// TwinCAT 3 PLC project OEF_6
// ProgramVersion: 3.1.4024.0
// libraries:
//   Tc2_BABasic, * (Beckhoff Automation GmbH)
//   Tc2_Standard, * (Beckhoff Automation GmbH)
//   Tc2_System, * (Beckhoff Automation GmbH)
//   Tc3_Module, * (Beckhoff Automation GmbH)
// project tree:
//   / PlcTask.TcTTO
//   POUs/ MAIN.TcPOU
// (motion and I/O tree: see PLC project oef_1)
// real-time tasks:
//   TASK PlcTask: cycle T#10ms, priority 20, ADS port 350
//   TASK PlcTask1: cycle T#10ms, priority 21, ADS port 351
//   TASK PlcTask2: cycle T#10ms, priority 22, ADS port 352
//   TASK PlcTask3: cycle T#10ms, priority 23, ADS port 353
//   TASK PlcTask4: cycle T#10ms, priority 24, ADS port 354
//   TASK PlcTask5: cycle T#10ms, priority 25, ADS port 355
//   TASK PlcTask6: cycle T#10ms, priority 26, ADS port 356
// variable links:
//   OEF_6/OEF_6 Instance <-> Device 1 (EtherCAT)/Term 1 (EK1200)/Term 3 (EL2008)
//     PlcTask Outputs/MAIN.buffer <-> Channel 1/Output
//     PlcTask Outputs/MAIN.buffer @bit 1 <-> Channel 2/Output
//     PlcTask Outputs/MAIN.buffer @bit 2 <-> Channel 3/Output
//     PlcTask Outputs/MAIN.buffer @bit 3 <-> Channel 4/Output
//   OEF_6/OEF_6 Instance <-> Device 1 (EtherCAT)/Term 1 (EK1200)/Term 4 (EL3062)
//     PlcTask Inputs/MAIN.Ninput <-> AI Standard Channel 1/Value

CONFIGURATION OEF_6
    RESOURCE PLC ON TwinCAT3
        TASK PlcTask(INTERVAL := T#10ms, PRIORITY := 25);
        PROGRAM MAIN WITH PlcTask : MAIN;
    END_RESOURCE
END_CONFIGURATION

// ---- POUs/MAIN.TcPOU
PROGRAM MAIN
VAR
	Ninput AT %I*: INT := 0;
	buffer AT %Q*: Byte := 0;
END_VAR

buffer := To_byte(F_Scale(Ninput,0,32767,0,15));

END_PROGRAM
